TYPE ST_ACswitchgear_IO :
STRUCT
	b_OutputMCCBShuntOk		AT %I* : BOOL;
	b_OutputMCCBfb			AT %I* : BOOL;
	b_penFb					AT %I* : BOOL;
	b_CEEprefuseOK			AT %I* : BOOL;
	b_Synchronizerfb		AT %I* : BOOL;
	b_InputMCCBfb			AT %I* : BOOL;
	b_InputContactorFb		AT %I* : BOOL;
	b_InputMCCBShuntOK		AT %I* : BOOL;
	b_InputContactorClose	AT %Q* : BOOL;
	b_InputContactorOpen	AT %Q* : BOOL;
	b_SyncEnable			AT %Q* : BOOL;

END_STRUCT
END_TYPE

(* stored: Version 1.1.0.1, ProductVersion 3.1.4026.18
   DUT ST_ACswitchgear_IO: Id {cedeb53f-8b44-4d49-b2b6-c06f7ef54e2e} *)
